// Mitsubishi GX Works2 project: Hil2   PLC: FX2N/FX2NC

// global labels: Global1
VAR_GLOBAL
  Verdiendring_1 : Verdiendring;
  Settpunkt_Kp_glob AT D2 : REAL;
  Settpunkt_Ki_glob AT D4 : REAL;
  Settpunkt_Kd_glob AT D6 : REAL;
  Settpunkt_Referanse_glob AT D0 : REAL;
  Tf_glob AT D8 : REAL;
  Tankp AT D10 : REAL;
  fP_glob AT D12 : REAL;
  fI_glob AT D14 : REAL;
  fDD AT D16 : REAL;
  Referanse_glob : INT;
  Kp_glob : REAL;
  Ki_glob : REAL;
  Kd_glob : REAL;
  Pådrag AT D20 : REAL;
  PID_REGULATOR_1 : PID_REGULATOR;
  fTs_glob AT D22 : REAL;
  fManOutput_glob : REAL;
END_VAR
VAR_GLOBAL CONSTANT
  fNomPådrag_glob : REAL := 0.04;
END_VAR

// task Task_01 (event TRUE, interval 0, priority 31): POU_01

FUNCTION_BLOCK PID_REGULATOR
VAR_INPUT
  referans : REAL;
  mea : REAL;
  fKp : REAL;
  fKi : REAL;
  fKd : REAL;
END_VAR
VAR_OUTPUT
  fOut : REAL;
  fP : REAL;
END_VAR
VAR
  fError : REAL;
END_VAR
VAR_OUTPUT
  fI : REAL;
END_VAR
VAR CONSTANT
  fTi : REAL := 10;
END_VAR
VAR
  fTs : REAL;
END_VAR
VAR_OUTPUT
  fD_term : REAL;
END_VAR
VAR
  fError_prev : REAL;
  fTracking : REAL;
END_VAR
VAR CONSTANT
  fNom : REAL := 0.04;
END_VAR
VAR
  bUseI : BOOL;
  bUseD : BOOL;
END_VAR
VAR_INPUT
  fTf : REAL;
END_VAR
VAR CONSTANT
  fTd : REAL := 1.0;
END_VAR
VAR
  fDfilter : REAL;
  fRawOut : REAL;
END_VAR
VAR_INPUT
  fFwd : REAL;
END_VAR
VAR
  bUseFwd : BOOL;
END_VAR
VAR_INPUT
  bMan : BOOL;
END_VAR
VAR
  fRef : REAL;
  fKt : REAL;
  fManOutput : REAL;
END_VAR
VAR CONSTANT
  fOutMax : REAL := 100.0;
END_VAR
VAR
  bSaturated : BOOL;
END_VAR
VAR CONSTANT
  fOutMin : REAL;
  input : BOOL := TRUE;
END_VAR
VAR_INPUT
  ManOutput : REAL;
  fKff : REAL;
  bForover : BOOL;
END_VAR
VAR
  bUseI_prev : BOOL;
  skan : INT;
  fskan : REAL;
  bInit : BOOL;
  bTimer : BOOL;
  bMan_prev : BOOL;
  bInitDone : BOOL;
END_VAR
fRef := referans;

(* Timer for fast eksekveringsfrekvens *)
bTimer := TRUE;
OUT_T(bTimer, TC0, 1);  (* 10ms *)

IF TS0 THEN
    bTimer := FALSE;
    fTs := 0.01;

    bUseI := fKi > 0.0;
    bUseD := fKd > 0.0;

    fError := fRef - mea;

    (* Rykkfri overgang til manuell *)
    IF bMan AND NOT bMan_prev THEN
        fManOutput_glob := fOut;
    END_IF;
    bMan_prev := bMan;

    (* P-ledd *)
    fP := fKp * fError;

    (* I-ledd *)
    IF bUseI THEN
        IF (NOT bUseI_prev) AND bInitDone THEN
            fI := fOut - fP - fD_term - (fFwd * fKff);
        ELSE
            fI := fI + fTs * (fKi * fError);
            IF fI > fOutMax THEN fI := fOutMax; END_IF;
            IF fI < fOutMin THEN fI := fOutMin; END_IF;
        END_IF;
    ELSE
        fI := fNomPådrag_glob;
    END_IF;
    bUseI_prev := bUseI;
    bInitDone := TRUE;

    (* D-ledd *)
    IF bUseD AND fTf > 0.0 THEN
        fDfilter := fDfilter + fTs / fTf * (fKd / fTs * (fError - fError_prev) - fDfilter);
        fD_term  := fDfilter;
    ELSE
        fD_term := 0.0;
    END_IF;

    (* Foroverkobling *)
    fRawOut := fP + fI + fD_term;
    IF bForover THEN
        fRawOut := fRawOut + (fFwd * fKff);
    END_IF;

    IF bMan THEN
        fOut := ManOutput;
        IF bForover THEN
            fI := ManOutput - fP - fD_term - (fFwd * fKff);
        ELSE
            fI := ManOutput - fP - fD_term;
        END_IF;
    ELSE
        (* Begrens output *)
        IF fRawOut > fOutMax THEN
            fOut       := fOutMax;
            bSaturated := TRUE;
        ELSIF fRawOut < fOutMin THEN
            fOut       := fOutMin;
            bSaturated := TRUE;
        ELSE
            fOut       := fRawOut;
            bSaturated := FALSE;
        END_IF;

        (* Anti-windup *)
        IF fKp > 0.0 THEN
            fKt := fKi / fKp;
        ELSE
            fKt := 0.0;
        END_IF;
        fTracking := fKt * (fOut - fRawOut);
    END_IF;

    fError_prev := fError;
    fTs_glob    := fTs;

END_IF;  (* TS0 *)
END_FUNCTION_BLOCK

PROGRAM POU_01
(* structured ladder/FBD written out as ST: instructions are called as NAME(EN, inputs, outputs); _pN, _eN, _tN stand for wires *)
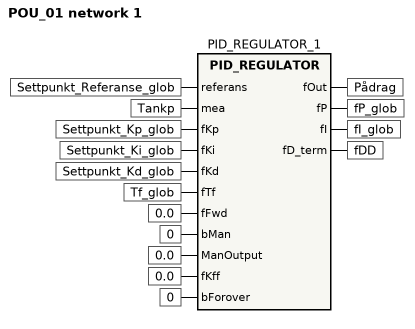
(* network 1 *)
PID_REGULATOR_1(referans := Settpunkt_Referanse_glob, mea := Tankp, fKp := Settpunkt_Kp_glob, fKi := Settpunkt_Ki_glob, fKd := Settpunkt_Kd_glob, fTf := Tf_glob, fFwd := 0.0, bMan := 0, ManOutput := 0.0, fKff := 0.0, bForover := 0, fOut => Pådrag, fP => fP_glob, fI => fI_glob, fD_term => fDD);
END_PROGRAM

FUNCTION_BLOCK Rampe
VAR_INPUT
  OldValue : REAL;
  NewValue : REAL;
END_VAR
VAR
  RampStep : REAL;
END_VAR
VAR_OUTPUT
  RampOut : REAL;
END_VAR
VAR
  rStartValue : REAL;
  rProgress : REAL;
  rLastTarget : REAL;
  rT_smooth : REAL;
END_VAR
VAR CONSTANT
  fRateSek : REAL := 5.0;
END_VAR


IF fRateSek > 0.0 THEN
	RampStep := 1.0 / (fRateSek * 100.0);
END_IF;

IF NewValue <> rLastTarget THEN
    rStartValue  := RampOut;
    rProgress    := 0.0;
    rLastTarget  := NewValue;
END_IF;

IF rProgress < 1.0 THEN
    rProgress := rProgress + RampStep;

    IF rProgress > 1.0 THEN
        rProgress := 1.0;
    END_IF;

    (*Smoothstep funksjon, formel: 3t² - 2t³ *)	
    rT_smooth := rProgress * rProgress * (3.0 - (2.0 * rProgress));

    RampOut := rStartValue + ((NewValue - rStartValue) * rT_smooth);
ELSE
    RampOut := NewValue;
END_IF;
END_FUNCTION_BLOCK

FUNCTION_BLOCK Verdiendring
VAR
  Rampe_1 : Rampe;
END_VAR
VAR_INPUT
  Settpunkt_Kp : REAL;
  Settpunkt_Ki : REAL;
  Settpunkt_Kd : REAL;
END_VAR
VAR_OUTPUT
  Kp : REAL;
  Ki : REAL;
  Kd : REAL;
  referanse : INT;
END_VAR
VAR_INPUT
  Settpunkt_referanse : INT;
END_VAR
VAR
  fSettpunkt_referanse : REAL;
  fReferanse : REAL;
  Rampe_2 : Rampe;
  Rampe_3 : Rampe;
  Rampe_4 : Rampe;
  iRateSek : INT;
END_VAR
(* structured ladder/FBD written out as ST: instructions are called as NAME(EN, inputs, outputs); _pN, _eN, _tN stand for wires *)
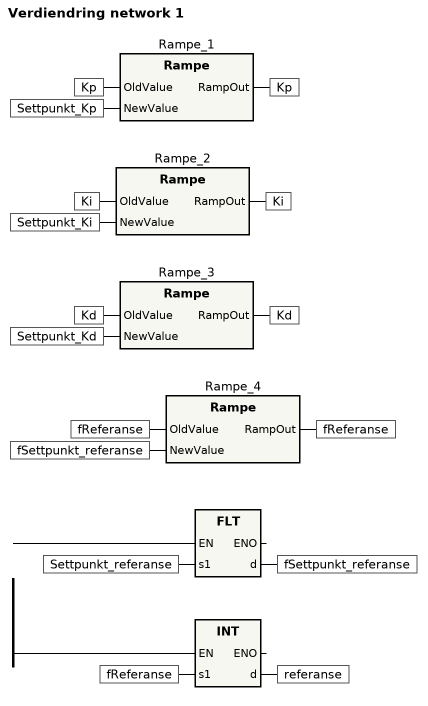
(* network 1 *)
Rampe_1(OldValue := Kp, NewValue := Settpunkt_Kp, RampOut => Kp);
Rampe_2(OldValue := Ki, NewValue := Settpunkt_Ki, RampOut => Ki);
Rampe_3(OldValue := Kd, NewValue := Settpunkt_Kd, RampOut => Kd);
Rampe_4(OldValue := fReferanse, NewValue := fSettpunkt_referanse, RampOut => fReferanse);
FLT(TRUE, Settpunkt_referanse, fSettpunkt_referanse);
INT(TRUE, fReferanse, referanse);
END_FUNCTION_BLOCK
